// TIA Portal V21 export
TYPE "coneCrusherConfig"
   STRUCT
      almMask : DWord := DW#16#FFFFFFFF;
      crushOutTime : Time := T#30s;
      premoldingDelay : Time := T#5s;
      premoldingClearTime : Time := T#30s;
      firstSignalTime : Time := T#10s;
      pauseSignalTime : Time := T#10s;
      secondSignalTime : Time := T#20s;
      soundFbDelay : Time := T#3s;
      signalTestTime : Time := T#10s;
      stopSignalStTime : Time := T#3s;
   END_STRUCT;
END_TYPE
